// TIA Portal V19 export
FUNCTION_BLOCK "RandomDataGenerator"   // FB2, LAD
{ S7_Optimized_Access := 'TRUE' }
// stored: MemoryReserve 100, SetENOAutomatically false
   VAR
      RandInt_1 : Int;
      RandInt_2 : Int;
      RandInt_3 : Int;
      RandInt_4 : Int;
      RandInt_5 : Int;
      RandReal_1 : Real;
      RandReal_2 : Real;
      RandReal_3 : Real;
      RandReal_4 : Real;
      RandReal_5 : Real;
   END_VAR
   VAR_TEMP
      Err : Array[0..9] of Bool;
      StatId : Array[0..9] of UInt;
      Stat : Array[0..9] of Word;
      i : USInt;
   END_VAR
BEGIN

REGION Network 1 (SCL)
   // Generowanie losowych danych
   #RandInt_1 := "LGF_RandomInt"(minValue:=0, maxValue:=1000, error=>#Err[0], statusID=>#StatId[0], status=>#Stat[0]);
   #RandInt_2 := "LGF_RandomInt"(minValue := 0, maxValue := 20, error => #Err[1], statusID => #StatId[1], status => #Stat[1]);
   #RandInt_3 := "LGF_RandomInt"(minValue := 0, maxValue := 30, error => #Err[2], statusID => #StatId[2], status => #Stat[2]);
   #RandInt_4 := "LGF_RandomInt"(minValue := -500, maxValue := 500, error => #Err[3], statusID => #StatId[3], status => #Stat[3]);
   #RandInt_5 := "LGF_RandomInt"(minValue := 1, maxValue := 8, error => #Err[4], statusID => #StatId[4], status => #Stat[4]);
   #RandReal_1 := "LGF_RandomReal"(minValue := 0.0, maxValue := 1000.0, error => #Err[5], statusID => #StatId[5], status => #Stat[5]);
   #RandReal_2 := "LGF_RandomReal"(minValue := 60.0, maxValue := 100.0, error => #Err[6], statusID => #StatId[6], status => #Stat[6]);
   #RandReal_3 := "LGF_RandomReal"(minValue := -30.0, maxValue := 30.0, error => #Err[7], statusID => #StatId[7], status => #Stat[7]);
   #RandReal_4 := "LGF_RandomReal"(minValue := 0.0, maxValue := 50.0, error => #Err[8], statusID => #StatId[8], status => #Stat[8]);
   #RandReal_5 := "LGF_RandomReal"(minValue := 0.0, maxValue := 6.28, error => #Err[9], statusID => #StatId[9], status => #Stat[9]);

   // Przepisanie do bloków _Interface wykorzystywanych w ćwiczeniach
   FOR #i := 0 TO 4 DO
       // Dla OPC
       "OPC_Interface".NumericalValues[#i] := #RandInt_1 * (#i + 1);
       "OPC_Interface".FloatingPointValues[#i] := #RandReal_1 / (#i + 1);
       "OPC_Interface".Booleans[#i] := "OPC_Interface".NumericalValues[#i].%X7;
       // Dla S7
       "S7_Interface".NumericalValues[#i] := 100 - #RandInt_2 - #i;
       "S7_Interface".FloatingPointValues[#i] := #RandReal_2 + (#i * 5);
       "S7_Interface".Booleans[#i] := "OPC_Interface".NumericalValues[#i].%X6;
   END_FOR;
END_REGION
END_FUNCTION_BLOCK
